PROGRAM MAIN
VAR
END_VAR

END_PROGRAM

(* stored: Version 1.1.0.1
   POU MAIN: Id {22f57513-1035-46b0-8179-c928d22964ce} *)
